# EPICS autosave request: CARSApp/Db/Energy_settings.req
# FILE... Energy_settings.req
$(P)$(EN):width.VAL
$(P)$(EN):dspace.VAL
$(P)$(EN):height.VAL
$(P)$(EN):id_off.VAL
$(P)$(EN):id_track.VAL
$(P)$(EN):use_id.VAL
$(P)$(EN):z2_track.VAL
$(P)$(EN):z2_off.VAL
$(P)$(EN):y2_track.VAL
$(P)$(EN):y2_off.VAL
$(P)$(EN):xt_track.VAL
$(P)$(EN):xt_sign.VAL
$(P)$(EN):xt_mvmin.VAL
$(P)$(EN):xt_off.VAL
$(P)$(EN):verbose.VAL
$(P)$(EN):tweakval.VAL
